KUKA KRL program: mh_lin_tr.src

&ACCESS RVP
&REL 2
&PARAM TEMPLATE = C:\KRC\Roboter\Template\vorgabe
&PARAM EDITMASK = *

; Main program
DEF mh_lin_tr( )

; DECL section

; Kuka's variables
STRUC str char s[81]
DECL str sendtext[9]
DECL str rectext[10]
DECL char sensorname[40]
DECL str dummy
BOOL errbl
BOOL brk
INT  errint
INT i
INT counter
FRAME extframe
BOOL bNew

; MH Variables
; prepending with mh because namespace is full of robot variables
INT mh_wait_seconds
BOOL mh_running
INT	mh_in_tick

INT	mh_mode
INT	mh_in_traject_id
INT	mh_out_traject_id

INT mh_robot_status
REAL mh_velocity
INT mh_framecount
INT mh_frameloop_counter
INT mh_tolerance

DECL STATE_T state

;BASISTECH INI
;GLOBAL INTERRUPT DECL 3 WHEN $STOPMESS==TRUE DO IR_STOPM ( )
;INTERRUPT ON 3

; ------------------------------------------------------------------
; BCO - PTP HOME
; Robot must do a BCO before anything else
; ------------------------------------------------------------------
BAS (#INITMOV,0 )
$BWDSTART=FALSE
PDAT_ACT=PDEFAULT
FDAT_ACT=FHOME
BAS(#PTP_PARAMS,30)
$H_POS=XHOME
PTP XHOME
; ------------------------------------------------------------------


;Init variables
brk = FALSE
counter = 0

mh_wait_seconds = 1
mh_running = TRUE
mh_in_tick = 0

errint = 0
mh_mode = 0
mh_in_traject_id = 0
mh_out_traject_id = 0

mh_robot_status = 0
mh_velocity = 200
mh_framecount = 1
mh_tolerance = 20

; receive structure
rectext[1].s[] = "Mateusz.ExternalData"
rectext[2].s[] = "Mateusz.ExternalData.Mode"
rectext[3].s[] = "Mateusz.ExternalData.Tick"
rectext[4].s[] = "Mateusz.ExternalData.Id"
rectext[5].s[] = "Mateusz.ExternalData.Run"
rectext[6].s[] = "Mateusz.ExternalData.Vel"
rectext[7].s[] = "Mateusz.ExternalData.Tol"
rectext[8].s[] = "Mateusz.ExternalData.Frames"
rectext[9].s[] = "Mateusz.ExternalData.XFrame"

;Open channel
sensorname[]="Mateusz"
errint = EKX_open(sensorname[])
EKX_handleerror(errint)

;Wait a little to let channel open
WAIT SEC mh_wait_seconds

; The channel is open and the server expect data from robot
; This is the very first message - telling that robot is ready.
mh_robot_status = 0 ; 0 means "Ready"
mh_out_traject_id = 0	; 0 means no trajectory, trajectory_id shall start at 1
mh_send_report()


$TIMER[1] = 0
$TIMER_STOP[1]=FALSE

; ------------------------------------------------------------------
; *** Main loop ***
; From now on robot waits for data, moves, and sends back reports
; ------------------------------------------------------------------
WHILE mh_running == TRUE

;Get Data from stack, only if there are new values

; The 0 means that we want next, not last (see krlxml.src)
; -1 means no timeout
errbl = EKX_WaitForSensorData(0, rectext[1].s[], -1)
IF errbl == FALSE THEN
   HALT
ENDIF

; get mode
errbl = EKX_GetIntegerElement(0, rectext[2].s[], mh_mode, bNew)
IF errbl == FALSE THEN
   HALT
ENDIF

; get tick
errbl = EKX_GetIntegerElement(0, rectext[3].s[], mh_in_tick, bNew)
IF errbl == FALSE THEN
   HALT
ENDIF

; get id
errbl = EKX_GetIntegerElement(0, rectext[4].s[], mh_in_traject_id, bNew)
IF errbl == FALSE THEN
   HALT
ENDIF

; get mh_running - a zero will terminate main loop after trajectory
errbl = EKX_GetBoolElement(0, rectext[5].s[], mh_running, bNew)
IF errbl == FALSE THEN
   HALT
ENDIF

; get velocity
errbl = EKX_GetRealElement(0, rectext[6].s[], mh_velocity, bNew)
IF errbl == FALSE THEN
   HALT
ENDIF

; set velocity for trajectory
$VEL.CP = (mh_velocity*0.001)

; get tolerance
errbl = EKX_GetIntegerElement(0, rectext[7].s[], mh_tolerance, bNew)
IF errbl == FALSE THEN
   HALT
ENDIF

; set tolerance for trajectory
$APO.CDIS=mh_tolerance

; get framecount
errbl = EKX_GetIntegerElement(0, rectext[8].s[], mh_framecount, bNew)
IF errbl == FALSE THEN
   HALT
ENDIF

; report that a message has been received
mh_robot_status = 1	; 1 means robot is about to execute a trajectory
mh_out_traject_id = mh_in_traject_id	; so we can tell which trajectory is received
mh_send_report()

; ---------------------------------
; Move loop
; Iterate all frames in this trajectory
; ---------------------------------
FOR mh_frameloop_counter = 1 TO mh_framecount STEP 1

; get frame
errbl = EKX_GetFrameElement( 0,  rectext[9].s[], extframe, bNew)
IF errbl == FALSE THEN
   HALT
ENDIF

; move with distance approximation
LIN extframe C_DIS

ENDFOR
; ---------------------------------
; End move loop
; ---------------------------------

; report that a trajectory has been received
mh_robot_status = 2	; 2 means robot finished executing a trajectory
mh_send_report()


ENDWHILE
; ------------------------------------------------------------------
; End of main loop
; We get here when mh_running is set to false
; ------------------------------------------------------------------

; final report
mh_robot_status = 3	; 3 means ending program
mh_out_traject_id = 0	; no trajectory
mh_send_report()

errbl = EKX_close(sensorname[])
IF errbl == FALSE THEN
  HALT
ENDIF

END	; end main program

; ------------------------------------------------------------------
; Subprograms
; ------------------------------------------------------------------


DEF mh_send_report()

errint = EKX_WriteInteger("Mateusz.Robot.Status", mh_robot_status)
EKX_handleerror(errint)

errint = EKX_WriteInteger("Mateusz.Robot.Error", errint)
EKX_handleerror(errint)

errint = EKX_WriteInteger("Mateusz.Robot.Mode", mh_mode)
EKX_handleerror(errint)

errint = EKX_WriteInteger("Mateusz.Robot.Tick", $TIMER[1])
EKX_handleerror(errint)

errint = EKX_WriteInteger("Mateusz.Robot.Id", mh_out_traject_id)
EKX_handleerror(errint)

errint = EKX_WriteReal("Mateusz.Robot.ActPos.X", $pos_act.x)
EKX_handleerror(errint)
errint = EKX_WriteReal("Mateusz.Robot.ActPos.Y", $pos_act.y)
EKX_handleerror(errint)
errint = EKX_WriteReal("Mateusz.Robot.ActPos.Z", $pos_act.z)
EKX_handleerror(errint)
errint = EKX_WriteReal("Mateusz.Robot.ActPos.A", $pos_act.a)
EKX_handleerror(errint)
errint = EKX_WriteReal("Mateusz.Robot.ActPos.B", $pos_act.b)
EKX_handleerror(errint)
errint = EKX_WriteReal("Mateusz.Robot.ActPos.C", $pos_act.c)
EKX_handleerror(errint)

; Send document
errint = EKX_Send("Mateusz")
EKX_handleerror(errint)

END
